// SIMATIC S7-200 project (STEP 7-Micro/WIN), CPU 224 REL 02.01

ORGANIZATION_BLOCK PRINCIPAL:OB1
TITLE=COMENTARIOS DEL PROGRAMA
BEGIN
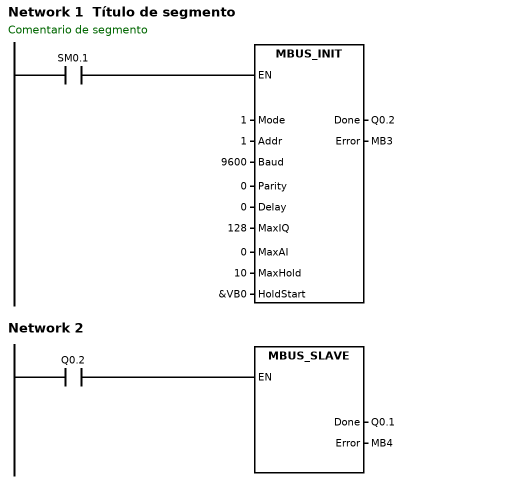
Network 1 // Título de segmento
// Comentario de segmento
LD     SM0.1
CALL   MBUS_INIT:SBR1, 1, 1, 9600, 0, 0, 128, 0, 10, &VB0, Q0.2, MB3
Network 2
LD     Q0.2
CALL   MBUS_SLAVE:SBR2, Q0.1, MB4
END_ORGANIZATION_BLOCK

// SBR1: protected block, not included

// SBR2: protected block, not included

// SBR3: protected block, not included
